FUNCTION_BLOCK FB_SimAxis
VAR_INPUT
END_VAR
VAR_OUTPUT
END_VAR
VAR
	fActPosition			AT %Q* : LREAL;
	fActVelocity			AT %Q* : LREAL;
	bReady					AT %Q* : BOOL := TRUE;
	bBusy					AT %Q* : BOOL;
	bError					AT %Q* : BOOL;
	bRunning				AT %Q* : BOOL;
	
	fPositionCmd			AT %I* : LREAL;
	fVelocityCmd			AT %I* : LREAL;
	bJogFwdCmd				AT %I* : BOOL;
	bMoveAbsCmd				AT %I* : BOOL;
	
	State					: DINT;
	fVelocity				: LREAL;
END_VAR

fVelocity := fVelocityCmd / 100.177;

CASE State OF
	0:
		bReady := TRUE;
		bBusy := FALSE;
		bError := FALSE;
		bRunning := FALSE;
		
		IF bJogFwdCmd THEN
			State := 10;
		END_IF
		
		IF bMoveAbsCmd AND (fActPosition <> fPositionCmd) THEN
			State := 20;
		END_IF
		
	10:
		bBusy := TRUE;
		bRunning := TRUE;
		bReady := FALSE;
		fActVelocity := fVelocityCmd;
		fActPosition := fActPosition + fVelocity;
		IF NOT bJogFwdCmd THEN
			State := 0;
		END_IF
		
	20:
		bBusy := TRUE;
		bRunning := TRUE;
		bReady := FALSE;
		IF fPositionCmd > fActPosition THEN
			State := 21;
		ELSE
			State := 22;
		END_IF
		
	21:
		IF (fPositionCmd > fActPosition) THEN
			fActPosition := fActPosition + fVelocity;
		ELSE
			fActPosition := fPositionCmd;
			State := 0;
		END_IF
		IF NOT bMoveAbsCmd THEN
			State := 0;
		END_IF
	
	22:
		fActVelocity := -(fVelocityCmd);
		IF (fPositionCmd < fActPosition) THEN
			fActPosition := fActPosition - fVelocity;
		ELSE
			fActPosition := fPositionCmd;
			State := 0;
		END_IF
		IF NOT bMoveAbsCmd THEN
			State := 0;
		END_IF
	
END_CASE

END_FUNCTION_BLOCK

(* stored: Version 1.1.0.1, ProductVersion 3.1.4024.12
   POU FB_SimAxis: Id {f89a4480-bdf9-4589-8e0d-cd64dcd27b44}, SpecialFunc None *)
